screen "System settings" 1280x740, template "Template_1"
   on GenerateScreen: SetTag("Tag_ScreenNumber", 5)
   Button "Calibrate screen" at 36,119 size 159x47; TextOff 'Calibrate screen'
      on Release: function_bc3e350c()
   Button "Clean screen" at 36,178 size 159x47; TextOff 'Clean screen'
      on Release: function_be740847(30)
   Button "Back" at 1,25 size 159x47; TextOff 'Back'
      on Release: ActivateScreen("System screens", 0)

screen "User administration" 1280x740, template "Template_1"
   on GenerateScreen: SetTag("Tag_ScreenNumber", 6)
   UserView "HmiScreenItemData" at 1,73 size 1197x659
   Button "Back" at 1,25 size 159x47; TextOff 'Back'
      on Release: ActivateScreen("System screens", 0)

screen "Different jobs" 1280x740, template "Template_1"
   on GenerateScreen: SetTag("Tag_ScreenNumber", 8)
   Button "Online" at 36,119 size 159x47; TextOff 'Online'
      on Release: function_bb44b551(0)
   Button "Offline" at 36,178 size 159x47; TextOff 'Offline'
      on Release: function_bb44b551(1)
   Button "Transfer" at 36,237 size 159x47; TextOff 'Transfer'
      on Release: function_bb44b551(2)
   Button "Toggle language" at 36,296 size 159x47; TextOff 'Toggle language'
      on Release: function_fb9197e8(-1)
   Button "Control Panel" at 36,355 size 159x47; TextOff 'Control Panel'
      on Release: function_f34a74f3()
   Button "Stop Runtime" at 36,414 size 159x47; TextOff 'Stop Runtime'
      on Release: StopRuntime(0)
   Button "Back" at 1,25 size 159x47; TextOff 'Back'
      on Release: ActivateScreen("System screens", 0)

screen "manual_mode" 1280x740, template "Template_1"
   on GenerateScreen: SetTag("Tag_ScreenNumber", 4)
   TrendView "Trend view_1" at 10,137 size 1188x595
   IOField "I/O field_1" at 317,63 size 137x63; FormatPattern 99999999999999999999
   TextField "Text field_1" at 62,71 size 269x46; Text 'Wartość zadana za pomocą potencjometru'

screen "automatic_mode" 1280x740, template "Template_1"
   on GenerateScreen: SetTag("Tag_ScreenNumber", 7)
   TrendView "Trend view_1" at 7,124 size 1184x601
   RecipeView "Recipe view_1" at 49,25 size 971x88; Recipe "Recipe_1"; Tag4DataRecord "RecipeNumber"
   Button "Button_1" at 1031,25 size 167x87; TextOff 'Załaduj Test'
      on Click: function_ac24277f("Recipe view_1")

screen "recipes" 1280x740, template "Template_1"
   on GenerateScreen: SetTag("Tag_ScreenNumber", 9)
   RecipeView "Recipe view_1" at 4,23 size 1176x704; DataRecordNameCaption 'Rodzaj testu:'; ValueCaption 'Wartość'; EntryNameCaption 'Parametr'; Recipe "Recipe_1"; Tag4DataRecord "RecipeNumber"

screen "Alarms" 1280x740, template "Template_1"
   on GenerateScreen: SetTag("Tag_ScreenNumber", 10)
   AlarmView "Alarm view_1" at 8,23 size 1176x709
*)